{attribute addProperty BoxType "EJ9576-0000-0018"}
{attribute addProperty Id "BCT_InputsAT %I*BCT_Inputs_7F924099128160WcStateAT %I*WcState_98A4DF7520.250InfoDataAT %I*InfoData_BC63D37F80100"}
{attribute addProperty CRC "3669577925"}
{attribute addProperty SizeInBites "210"}
{attribute addProperty SizeInBytes "26.25"}
TYPE EJ9576_30D5723B :
STRUCT
	{attribute addProperty Name "BCT_Inputs"}
	BCT_Inputs : BCT_Inputs_7F924099;
	{attribute addProperty Name "WcState"}
	WcState : WcState_98A4DF75;
	{attribute addProperty Name "InfoData"}
	InfoData : InfoData_BC63D37F;
END_STRUCT
END_TYPE

(* stored: Version 1.2.0.0, ProductVersion 3.1.4024.9
   DUT EJ9576_30D5723B: Id {c1ab1060-6267-43ad-9c9e-7176977b6656} *)
